// TIA Portal V17 export
// export: Created 2025-11-19T10:30:00.000Z, ExportSetting WithDefaults, DisplayName Totally Integrated Automation Portal, DisplayVersion V17
DATA_BLOCK "DB_GlobalData"   // DB1
{ S7_Optimized_Access := 'TRUE' }
VERSION : 0.1
// stored: AutoNumber true, DBAccessibleFromOPCUA true, DataBlockType GlobalDB, IsIECCheckEnabled false, IsRetainMemResEnabled false, MemoryReserve 100
   VAR
      Start_Button { ExternalWritable := 'False'} : Bool;   // Start button input
      Stop_Button : Bool;   // Stop button input
      Emergency_Stop : Bool;   // Emergency stop input
      Motor_Running : Bool;   // Motor running status
      Motor_Speed : Real := 0.0;   // Current motor speed RPM
      Speed_Setpoint : Real := 1500.0;   // Desired motor speed RPM
      Temperature : Real := 25.0;   // Motor temperature in Celsius
      RunTime_Hours : DInt := 0;   // Total runtime hours
      Alarm_Active : Bool;   // Alarm status flag
      Alarm_Code : Word := 16#0000;   // Alarm code identifier
   END_VAR
BEGIN
END_DATA_BLOCK
